FUNCTION_BLOCK Teste01 (* Template for a Basic Function Block Type *)
  (* Standard: 61499-2 *)
  (* Version 1.0, 2024-12-17, Bruno *)
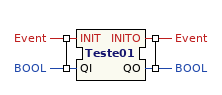
  EVENT_INPUT
    INIT WITH QI; (* Initialization Request *)
  END_EVENT
  EVENT_OUTPUT
    INITO WITH QO; (* Initialization Confirm *)
  END_EVENT
  VAR_INPUT
    QI : BOOL; (* Input event qualifier *)
  END_VAR
  VAR_OUTPUT
    QO : BOOL; (* Output event qualifier *)
  END_VAR
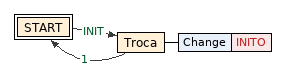
  EC_STATES
    START; (* Initial State *)
    Troca : Change -> INITO;
  END_STATES
  EC_TRANSITIONS
    START TO Troca := INIT;
    Troca TO START := 1;
  END_TRANSITIONS
  ALGORITHM Change IN ST:
QO :=  NOT QO;
  END_ALGORITHM
END_FUNCTION_BLOCK
